(* CoDeSys 2.3.9.55 project: AccesoRecinto.pro *)
(* Libraries: Standard.lib 2.6.14 10:37:46 *)

(* Global variable list: Global_Variables *)
VAR_GLOBAL
      (* Entradas*)
	A: BOOL;
	B: BOOL;

       (* Salidas*)
	LuzVerde: BOOL;
	LuzAmarilla: BOOL;
	LuzRoja: BOOL;

       (* Contador de la visualización *)
	Contador: CTUD;
END_VAR

(* POU PLC_PRG, ST *)
PROGRAM PLC_PRG
VAR
END_VAR

END_PROGRAM

(* Visualisation Teatro
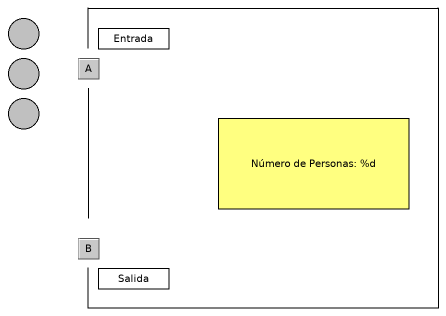
button at (120,80)-(141,101): text "A"; taps A
button at (120,260)-(141,281): text "B"; taps B
ellipse at (50,40)-(81,71): alarm colour if LuzRoja
ellipse at (50,80)-(81,111): alarm colour if LuzAmarilla
ellipse at (50,120)-(81,151): alarm colour if LuzVerde
rectangle at (260,140)-(451,231): text "Número de Personas: %d"; shows contador.CV
rectangle at (140,50)-(211,71): text "Entrada"
rectangle at (140,290)-(211,311): text "Salida"
2 more shapes without text or variables
*)
